FUNCTION Fill_Row_Two : BOOL
VAR_INPUT
	row: ARRAY [1..10] OF WORD;
END_VAR
VAR
END_VAR

GV_MODBUS.twoLeft[1]:= row[1];
GV_MODBUS.twoLeft[2]:= row[2];
GV_MODBUS.twoLeft[3]:= row[3];
GV_MODBUS.twoLeft[4]:= row[4];
GV_MODBUS.twoLeft[5]:= row[5];
GV_MODBUS.twoRight[1]:= row[6];
GV_MODBUS.twoRight[2]:= row[7];
GV_MODBUS.twoRight[3]:= row[8];
GV_MODBUS.twoRight[4]:= row[9];
GV_MODBUS.twoRight[5]:= row[10];

Fill_Row_Two := TRUE;

END_FUNCTION

(* stored: Version 1.1.0.1, ProductVersion 3.1.4022.12
   POU Fill_Row_Two: Id {3a251f3e-0781-4a93-9af1-89324f6e2c79}, SpecialFunc None *)
